FUNCTION_BLOCK EL2535
VAR
	{attribute addProperty Name "WcState"}
	_wcState : WcStateInputToggle;
	{attribute addProperty Name "Info data"}
	_infoData : InfoDataAds;
	_io : EL2535_Data;
END_VAR

PROPERTY IO : REFERENCE TO EL2535_Data
GET
IO REF= _io;
END_GET
END_PROPERTY

PROPERTY WcState : REFERENCE TO WcStateInputToggle
GET
WcState REF= _wcState;
END_GET
END_PROPERTY

END_FUNCTION_BLOCK

(* stored: Version 1.1.0.1, ProductVersion 3.1.4024.9
   POU EL2535: Id {15b0cd20-459b-0dfa-0a78-03aa88476959}, SpecialFunc None
   Property IO: Id {ea0f70b2-35b3-0719-2d17-16655dde4301}
   Get Get: Id {2abf4451-f793-0c1e-1945-8991e67edd7f}
   Property WcState: Id {f8160de3-2962-0972-3b9c-37da7e94b237}
   Get Get: Id {1f9a47e0-bcc4-05c6-14c7-8a9788f73e60} *)
